// TIA Portal V17 export
// export: Created 2026-04-13T11:12:54.4239411Z, ExportSetting WithDefaults, DisplayName Totally Integrated Automation Portal, DisplayVersion V17 Update 4, DisplayName TIA Portal Openness, DisplayVersion V17 Update 4, DisplayName TIA Portal Version Control Interface, DisplayVersion V17, DisplayName SINAMICS Startdrive Advanced, DisplayVersion V17, DisplayName SINAMICS Startdrive G130, G150, S120, S150, SINAMICS MV, S210, DisplayVersion V17, DisplayName SINAMICS Startdrive G110M, G120, G120C, G120D, G120P, G115D, DisplayVersion V17, DisplayName STEP 7 Professional, DisplayVersion V17 Update 4, DisplayName STEP 7 Safety, DisplayVersion V17, DisplayName WinCC Professional, DisplayVersion V17 Update 4
TagTable "操作日志"
  Audit_编号1 : WString  (1 s)
  Audit_编号2 : WString  (1 s)
  Audit_编号3 : WString  (1 s)
  Audit_编号4 : WString  (1 s)
  Audit_编号5 : WString  (1 s)
  Audit_编号6 : WString  (1 s)
  Audit_编号7 : WString  (1 s)
  Audit_编号8 : WString  (1 s)
  Audit_编号9 : WString  (1 s)
  Audit_编号10 : WString  (1 s)
  Audit_编号11 : WString  (1 s)
  Audit_编号12 : WString  (1 s)
  Audit_编号13 : WString  (1 s)
  Audit_编号14 : WString  (1 s)
  Audit_编号15 : WString  (1 s)
  Audit_时间1 : WString  (1 s)
  Audit_时间2 : WString  (1 s)
  Audit_时间3 : WString  (1 s)
  Audit_时间4 : WString  (1 s)
  Audit_时间5 : WString  (1 s)
  Audit_时间6 : WString  (1 s)
  Audit_时间7 : WString  (1 s)
  Audit_时间8 : WString  (1 s)
  Audit_时间9 : WString  (1 s)
  Audit_时间10 : WString  (1 s)
  Audit_时间11 : WString  (1 s)
  Audit_时间12 : WString  (1 s)
  Audit_时间13 : WString  (1 s)
  Audit_时间14 : WString  (1 s)
  Audit_时间15 : WString  (1 s)
  Audit_用户1 : WString  (1 s)
  Audit_用户2 : WString  (1 s)
  Audit_用户3 : WString  (1 s)
  Audit_用户4 : WString  (1 s)
  Audit_用户5 : WString  (1 s)
  Audit_用户6 : WString  (1 s)
  Audit_用户7 : WString  (1 s)
  Audit_用户8 : WString  (1 s)
  Audit_用户9 : WString  (1 s)
  Audit_用户10 : WString  (1 s)
  Audit_用户11 : WString  (1 s)
  Audit_用户12 : WString  (1 s)
  Audit_用户13 : WString  (1 s)
  Audit_用户14 : WString  (1 s)
  Audit_用户15 : WString  (1 s)
  Audit_对象1 : WString  (1 s)
  Audit_对象2 : WString  (1 s)
  Audit_对象3 : WString  (1 s)
  Audit_对象4 : WString  (1 s)
  Audit_对象5 : WString  (1 s)
  Audit_对象6 : WString  (1 s)
  Audit_对象7 : WString  (1 s)
  Audit_对象8 : WString  (1 s)
  Audit_对象9 : WString  (1 s)
  Audit_对象10 : WString  (1 s)
  Audit_对象11 : WString  (1 s)
  Audit_对象12 : WString  (1 s)
  Audit_对象13 : WString  (1 s)
  Audit_对象14 : WString  (1 s)
  Audit_对象15 : WString  (1 s)
  Audit_描述1 : WString  (1 s)
  Audit_描述2 : WString  (1 s)
  Audit_描述3 : WString  (1 s)
  Audit_描述4 : WString  (1 s)
  Audit_描述5 : WString  (1 s)
  Audit_描述6 : WString  (1 s)
  Audit_描述7 : WString  (1 s)
  Audit_描述8 : WString  (1 s)
  Audit_描述9 : WString  (1 s)
  Audit_描述10 : WString  (1 s)
  Audit_描述11 : WString  (1 s)
  Audit_描述12 : WString  (1 s)
  Audit_描述13 : WString  (1 s)
  Audit_描述14 : WString  (1 s)
  Audit_描述15 : WString  (1 s)
  执行说明 : WString  (1 s)
  日志当前页数 : Int  (1 s)
  日志总页数 : Int  (1 s)
